RoboDK station: soldagem_caixa.rdk

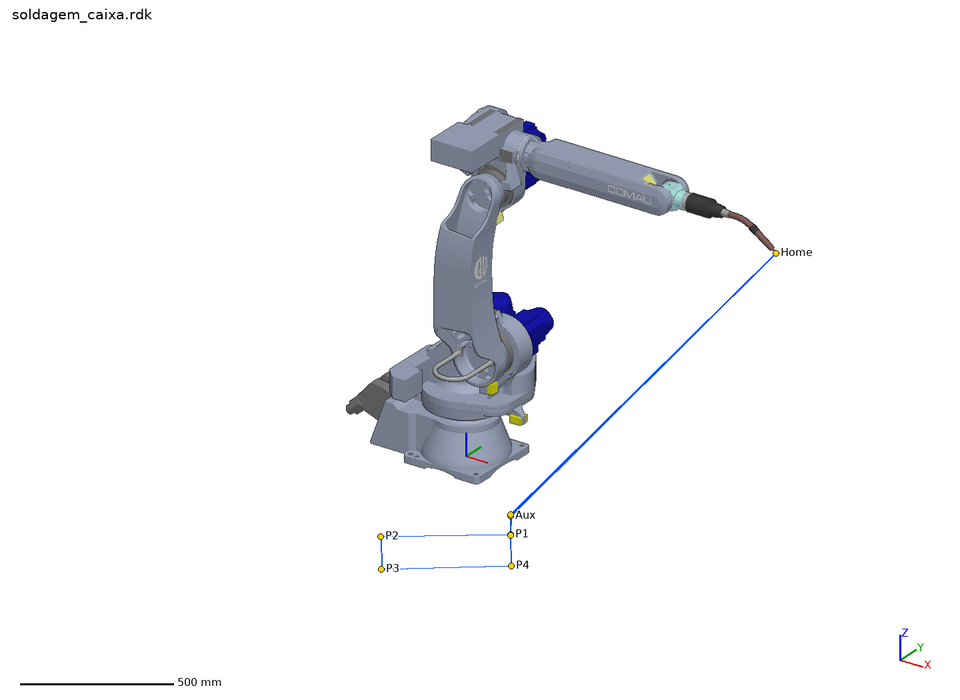
[picture v0: the station drawn from its stored meshes, robots at their saved joint values, targets as dots, program paths as lines]
Station soldagem_caixa (saved by RoboDK 5.6.4). Poses are relative to the parent item; angles as X-Y-Z fixed-axis rotations.
  - frame Comau Smart SiX 6-1.4 Base at (0, 0, 0) mm
    - robot Comau Smart SiX 6-1.4: 6 axes, payload 6 kg, reach 1400 mm, repeatability 0.05 mm, weight 160 kg
        modified DH rows (alpha deg, a mm, theta deg, d mm): 0, 0, 0, 450; -90, 150, -90, 0; 0, 590, -90, 0; -90, 130, 0, 647.07; 90, 0, 0, 0; -90, 0, 180, 95
        joint limits [-170, -85, -170, -210, -130, -400] to [170, 155, 0, 210, 130, 500]; home [0, 0, -90, 0, 0, 0]; saved at [0, 0, -90, 0, 0, 0]
      - tool Generic Welding Gun (Through-arm), TCP at (89, 0, 340) mm, rotated rx 0 ry 35 rz 0 deg, size 122.1 x 64 x 340.8 mm
    - target Home (joint target) at (1232.07, 0, 1081) mm, rotated rx -180 ry 55 rz -180 deg; joints [0, 0, -90, 0, 0, 0] of Comau Smart SiX 6-1.4
    - target Aux (joint target) at (678.19, -714.38, 259.33) mm, rotated rx -180 ry -35 rz -98.83 deg; joints [42.16, 19.904, -109.512, -0.001, 50.583, 123.333] of Comau Smart SiX 6-1.4
    - target P1 (joint target) at (674.01, -710.6, 189.6) mm, rotated rx -180 ry -35 rz -98.83 deg; joints [42.16, 22.966, -112.348, -0.001, 44.685, 123.334] of Comau Smart SiX 6-1.4
    - target P2 (joint target) at (337.62, -965.5, 189.61) mm, rotated rx -180 ry -35 rz -5.51 deg; joints [75.414, 28.001, -105.01, -0.002, 46.989, 249.903] of Comau Smart SiX 6-1.4
    - target P3 (joint target) at (476.07, -1160.5, 189.6) mm, rotated rx 180 ry -35 rz 85.86 deg; joints [69.397, 63.948, -44.768, -0.001, 71.283, 335.258] of Comau Smart SiX 6-1.4
    - target P4 (joint target) at (809.33, -897.92, 189.6) mm, rotated rx -180 ry -35 rz 172.67 deg; joints [45.37, 55.629, -59.624, -0.001, 64.746, 398.042] of Comau Smart SiX 6-1.4
    - target P1' (joint target) at (676.67, -711.86, 189.6) mm, rotated rx 180 ry -35 rz -107.27 deg; joints [41.72, 24.14, -110.67, 0, 45.19, 474.45] of Comau Smart SiX 6-1.4
    - target Aux' (joint target) at (676.65, -711.85, 264.02) mm, rotated rx -180 ry -35 rz -107.27 deg; joints [41.72, 20.44, -108.33, 0, 51.23, 474.45] of Comau Smart SiX 6-1.4
  - program Soldagem_Caixa_1_G1 (11 instructions, listed below)
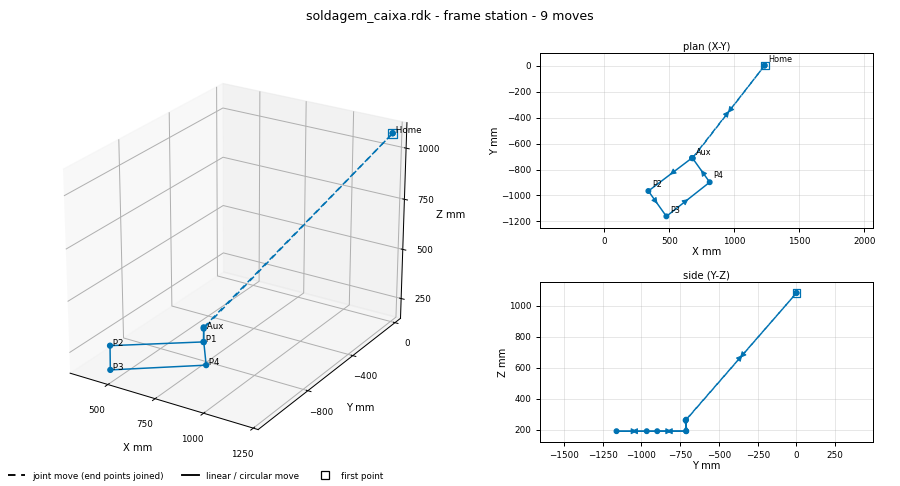
[picture p0: tool path of soldagem_caixa.rdk in frame station, 9 of 9 moves have a stored position in this frame; points joined in program order, loops and branches not executed]

--- program Soldagem_Caixa_1_G1 (robot Comau Smart SiX 6-1.4) ---
  Set Ref.: Comau Smart SiX 6-1.4 Base
  Set Tool: Generic Welding Gun (Through-arm)
  MoveJ (Target 1) -> target Home
  MoveJ (Target 2) -> target Aux
  MoveL (Target 3) -> target P1
  MoveL (Target 4) -> target P2
  MoveL (Target 5) -> target P3
  MoveL (Target 6) -> target P4
  MoveL (Target 7) -> target P1'
  MoveL (Target 8) -> target Aux'
  MoveJ (Home)
